(* IEC 61131-3 sources: com.logicals.lc3.webinar/usRTS_RPMControl_iSOC/src_FB_LIB_SAFE/Bitstring/BOOL, 10 files *)

(* ---- wAND_BOOL_2.iecst ---- *)
NAMESPACE logicals.web.standard
NAMESPACE bitstring

/*
 * Function block wrapper for IEC 61131-3 AND<br>
 * IN1 =  1st value (BOOL)<br>
 * IN2 =  2nd value (BOOL)<br>
 * OUT = IN1 AND IN2 (BOOL)<br>
 */
FUNCTION_BLOCK wAND_BOOL_2
	{ vNameAlignment:="center"; altName:="&"; bgColor:="MediumBlue"; width:=40; hideIONames; }
	VAR_INPUT
		IN1 : BOOL;
		IN2 : BOOL;
	END_VAR
	VAR_OUTPUT
		OUT: BOOL;
	END_VAR

	OUT := AND(IN1:=IN1, IN2:=IN2, ENO=>ENO);
END_FUNCTION_BLOCK

END_NAMESPACE
END_NAMESPACE

(* ---- wAND_BOOL_3.iecst ---- *)
NAMESPACE logicals.web.standard
NAMESPACE bitstring

/*
 * Function block wrapper for IEC 61131-3 AND<br>
 * IN1 =  1st value (BOOL)<br>
 * IN2 =  2nd value (BOOL)<br>
 * IN3 =  3rd value (BOOL)<br>
 * OUT = IN1 AND IN2 AND IN3 (BOOL)<br>
 */
FUNCTION_BLOCK wAND_BOOL_3
	{ vNameAlignment:="center"; altName:="&"; bgColor:="MediumBlue"; width:=40; hideIONames; }
	VAR_INPUT
		IN1 : BOOL;
		IN2 : BOOL;
		IN3 : BOOL;
	END_VAR
	VAR_OUTPUT
		OUT: BOOL;
	END_VAR

	OUT := AND(IN1:=IN1, IN2:=IN2, IN3:=IN3, ENO=>ENO);
END_FUNCTION_BLOCK

END_NAMESPACE
END_NAMESPACE

(* ---- wAND_BOOL_4.iecst ---- *)
NAMESPACE logicals.web.standard
NAMESPACE bitstring

/*
 * Function block wrapper for IEC 61131-3 AND<br>
 * IN1 =  1st value (BOOL)<br>
 * IN2 =  2nd value (BOOL)<br>
 * IN3 =  3rd value (BOOL)<br>
 * IN4 =  4th value (BOOL)<br>
 * OUT = IN1 AND IN2 AND IN3 AND IN4 (BOOL)<br>
 */
FUNCTION_BLOCK wAND_BOOL_4
	{ vNameAlignment:="center"; altName:="&"; bgColor:="MediumBlue"; width:=40; hideIONames; }
	VAR_INPUT
		IN1 : BOOL;
		IN2 : BOOL;
		IN3 : BOOL;
		IN4 : BOOL;
	END_VAR
	VAR_OUTPUT
		OUT: BOOL;
	END_VAR

	OUT := AND(IN1:=IN1, IN2:=IN2, IN3:=IN3, IN4:=IN4, ENO=>ENO);
END_FUNCTION_BLOCK

END_NAMESPACE
END_NAMESPACE

(* ---- wNOT_BOOL.iecst ---- *)
NAMESPACE logicals.web.standard
NAMESPACE bitstring

/*
 * Function block wrapper for IEC 61131-3 NOT<br>
 * IN = input (BOOL)<br>
 * OUT = !IN (BOOL)<br>
 */
FUNCTION_BLOCK wNOT_BOOL
	{ vNameAlignment:="center"; altName:="NOT"; bgColor:="MediumBlue"; width:=60; hideIONames; }
	VAR_INPUT
		IN : BOOL;
	END_VAR
	VAR_OUTPUT
		OUT: BOOL;
	END_VAR

	OUT := NOT(IN:=IN, ENO=>ENO);
END_FUNCTION_BLOCK

END_NAMESPACE
END_NAMESPACE

(* ---- wOR_BOOL_2.iecst ---- *)
NAMESPACE logicals.web.standard
NAMESPACE bitstring

/*
 * Function block wrapper for IEC 61131-3 OR<br>
 * IN1 =  1st value (BOOL)<br>
 * IN2 =  2nd value (BOOL)<br>
 * OUT = IN1 OR IN2 (BOOL)<br>
 */
FUNCTION_BLOCK wOR_BOOL_2
	{ vNameAlignment:="center"; altName:=">=1"; bgColor:="MediumBlue"; width:=40; hideIONames; }
	VAR_INPUT
		IN1 : BOOL;
		IN2 : BOOL;
	END_VAR
	VAR_OUTPUT
		OUT: BOOL;
	END_VAR

	OUT := OR(IN1:=IN1, IN2:=IN2, ENO=>ENO);
END_FUNCTION_BLOCK

END_NAMESPACE
END_NAMESPACE

(* ---- wOR_BOOL_3.iecst ---- *)
NAMESPACE logicals.web.standard
NAMESPACE bitstring

/*
 * Function block wrapper for IEC 61131-3 OR<br>
 * IN1 =  1st value (BOOL)<br>
 * IN2 =  2nd value (BOOL)<br>
 * IN3 =  3rd value (BOOL)<br>
 * OUT = IN1 OR IN2 OR IN3 (BOOL)<br>
 */
FUNCTION_BLOCK wOR_BOOL_3
	{ vNameAlignment:="center"; altName:=">=1"; bgColor:="MediumBlue"; width:=40; hideIONames; }
	VAR_INPUT
		IN1 : BOOL;
		IN2 : BOOL;
		IN3 : BOOL;
	END_VAR
	VAR_OUTPUT
		OUT: BOOL;
	END_VAR

	OUT := OR(IN1:=IN1, IN2:=IN2, IN3:=IN3, ENO=>ENO);
END_FUNCTION_BLOCK

END_NAMESPACE
END_NAMESPACE

(* ---- wOR_BOOL_4.iecst ---- *)
NAMESPACE logicals.web.standard
NAMESPACE bitstring

/*
 * Function block wrapper for IEC 61131-3 OR<br>
 * IN1 =  1st value (BOOL)<br>
 * IN2 =  2nd value (BOOL)<br>
 * IN3 =  3rd value (BOOL)<br>
 * IN4 =  4th value (BOOL)<br>
 * OUT = IN1 OR IN2 OR IN3 OR IN4 (BOOL)<br>
 */
FUNCTION_BLOCK wOR_BOOL_4
	{ vNameAlignment:="center"; altName:=">=1"; bgColor:="MediumBlue"; width:=40; hideIONames; }
	VAR_INPUT
		IN1 : BOOL;
		IN2 : BOOL;
		IN3 : BOOL;
		IN4 : BOOL;
	END_VAR
	VAR_OUTPUT
		OUT: BOOL;
	END_VAR

	OUT := OR(IN1:=IN1, IN2:=IN2, IN3:=IN3, IN4:=IN4, ENO=>ENO);
END_FUNCTION_BLOCK

END_NAMESPACE
END_NAMESPACE

(* ---- wXOR_BOOL_2.iecst ---- *)
NAMESPACE logicals.web.standard
NAMESPACE bitstring

/*
 * Function block wrapper for IEC 61131-3 XOR<br>
 * IN1 =  1st value (BOOL)<br>
 * IN2 =  2nd value (BOOL)<br>
 * OUT = IN1 XOR IN2 (BOOL)<br>
 */
FUNCTION_BLOCK wXOR_BOOL_2
	{ vNameAlignment:="center"; altName:="=2k+1"; bgColor:="MediumBlue"; width:=50; hideIONames; }
	VAR_INPUT
		IN1 : BOOL;
		IN2 : BOOL;
	END_VAR
	VAR_OUTPUT
		OUT: BOOL;
	END_VAR

	OUT := XOR(IN1:=IN1, IN2:=IN2, ENO=>ENO);
END_FUNCTION_BLOCK

END_NAMESPACE
END_NAMESPACE

(* ---- wXOR_BOOL_3.iecst ---- *)
NAMESPACE logicals.web.standard
NAMESPACE bitstring

/*
 * Function block wrapper for IEC 61131-3 XOR<br>
 * IN1 =  1st value (BOOL)<br>
 * IN2 =  2nd value (BOOL)<br>
 * IN3 =  3rd value (BOOL)<br>
 * OUT = IN1 XOR IN2 XOR IN3 (BOOL)<br>
 */
FUNCTION_BLOCK wXOR_BOOL_3
	{ vNameAlignment:="center"; altName:="=2k+1"; bgColor:="MediumBlue"; width:=50; hideIONames; }
	VAR_INPUT
		IN1 : BOOL;
		IN2 : BOOL;
		IN3 : BOOL;
	END_VAR
	VAR_OUTPUT
		OUT: BOOL;
	END_VAR

	OUT := XOR(IN1:=IN1, IN2:=IN2, IN3:=IN3, ENO=>ENO);
END_FUNCTION_BLOCK

END_NAMESPACE
END_NAMESPACE

(* ---- wXOR_BOOL_4.iecst ---- *)
NAMESPACE logicals.web.standard
NAMESPACE bitstring

/*
 * Function block wrapper for IEC 61131-3 XOR<br>
 * IN1 =  1st value (BOOL)<br>
 * IN2 =  2nd value (BOOL)<br>
 * IN3 =  3rd value (BOOL)<br>
 * IN4 =  4th value (BOOL)<br>
 * OUT = IN1 XOR IN2 XOR IN3 XOR IN4 (BOOL)<br>
 */
FUNCTION_BLOCK wXOR_BOOL_4
	{ vNameAlignment:="center"; altName:="=2k+1"; bgColor:="MediumBlue"; width:=50; hideIONames; }
	VAR_INPUT
		IN1 : BOOL;
		IN2 : BOOL;
		IN3 : BOOL;
		IN4 : BOOL;
	END_VAR
	VAR_OUTPUT
		OUT: BOOL;
	END_VAR

	OUT := XOR(IN1:=IN1, IN2:=IN2, IN3:=IN3, IN4:=IN4, ENO=>ENO);
END_FUNCTION_BLOCK

END_NAMESPACE
END_NAMESPACE
